FUNCTION_BLOCK FC_Occupation (* Free / Occupied / Priority / Local; trusted operator boundary; release/override only when quiescent *)
  (* Standard: 61499-2 *)
  (* Version 2.0, 2026-09-27, Project contributors, Filling cell reference model *)
  PACKAGE fillingcell;
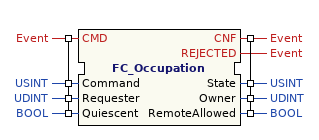
  EVENT_INPUT
    CMD WITH Command, Requester, Quiescent;
  END_EVENT
  EVENT_OUTPUT
    CNF WITH State, Owner, RemoteAllowed;
    REJECTED;
  END_EVENT
  VAR_INPUT
    Command : USINT;
    Requester : UDINT;
    Quiescent : BOOL;
  END_VAR
  VAR_OUTPUT
    State : USINT;
    Owner : UDINT;
    RemoteAllowed : BOOL;
  END_VAR
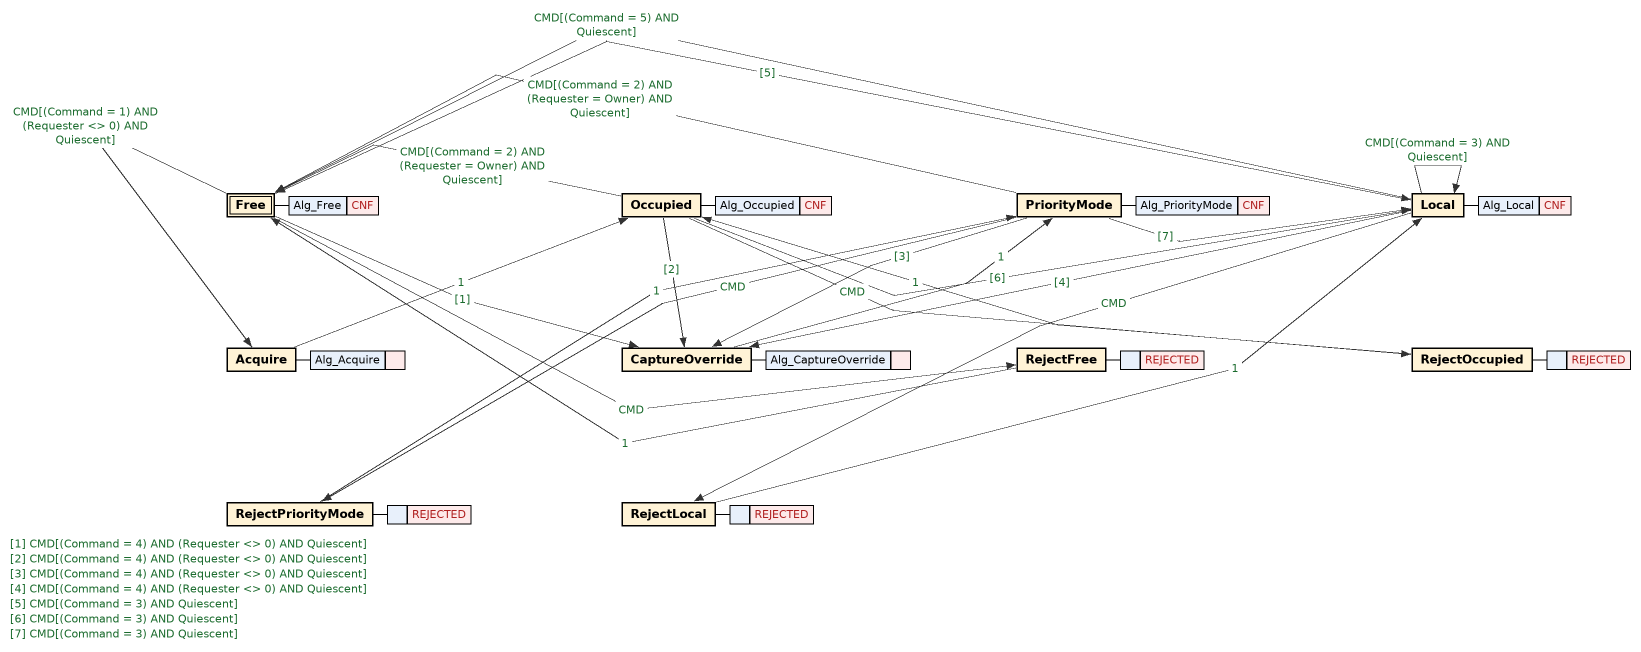
  EC_STATES
    Free : Alg_Free -> CNF;
    Occupied : Alg_Occupied -> CNF;
    PriorityMode : Alg_PriorityMode -> CNF;
    Local : Alg_Local -> CNF;
    Acquire : Alg_Acquire;
    CaptureOverride : Alg_CaptureOverride;
    RejectFree : -> REJECTED;
    RejectOccupied : -> REJECTED;
    RejectPriorityMode : -> REJECTED;
    RejectLocal : -> REJECTED;
  END_STATES
  EC_TRANSITIONS
    Free TO Acquire := CMD[(Command = 1) AND (Requester <> 0) AND Quiescent];
    Occupied TO Free := CMD[(Command = 2) AND (Requester = Owner) AND Quiescent];
    PriorityMode TO Free := CMD[(Command = 2) AND (Requester = Owner) AND Quiescent];
    Local TO Free := CMD[(Command = 5) AND Quiescent];
    Free TO Local := CMD[(Command = 3) AND Quiescent];
    Free TO CaptureOverride := CMD[(Command = 4) AND (Requester <> 0) AND Quiescent];
    Free TO RejectFree := CMD;
    RejectFree TO Free := 1;
    Occupied TO Local := CMD[(Command = 3) AND Quiescent];
    Occupied TO CaptureOverride := CMD[(Command = 4) AND (Requester <> 0) AND Quiescent];
    Occupied TO RejectOccupied := CMD;
    RejectOccupied TO Occupied := 1;
    PriorityMode TO Local := CMD[(Command = 3) AND Quiescent];
    PriorityMode TO CaptureOverride := CMD[(Command = 4) AND (Requester <> 0) AND Quiescent];
    PriorityMode TO RejectPriorityMode := CMD;
    RejectPriorityMode TO PriorityMode := 1;
    Local TO Local := CMD[(Command = 3) AND Quiescent];
    Local TO CaptureOverride := CMD[(Command = 4) AND (Requester <> 0) AND Quiescent];
    Local TO RejectLocal := CMD;
    RejectLocal TO Local := 1;
    Acquire TO Occupied := 1;
    CaptureOverride TO PriorityMode := 1;
  END_TRANSITIONS
  ALGORITHM Alg_Free IN ST:
State := 0;
RemoteAllowed := FALSE;
Owner := 0;
  END_ALGORITHM
  ALGORITHM Alg_Occupied IN ST:
State := 1;
RemoteAllowed := TRUE;
  END_ALGORITHM
  ALGORITHM Alg_PriorityMode IN ST:
State := 2;
RemoteAllowed := TRUE;
  END_ALGORITHM
  ALGORITHM Alg_Local IN ST:
State := 3;
RemoteAllowed := FALSE;
Owner := 0;
  END_ALGORITHM
  ALGORITHM Alg_Acquire IN ST:
Owner := Requester;
  END_ALGORITHM
  ALGORITHM Alg_CaptureOverride IN ST:
Owner := Requester;
  END_ALGORITHM
END_FUNCTION_BLOCK
